ABB RAPID module: Module1

MODULE Module1

    CONST robtarget BackFromStop:=[[674.324181213,-18.678370802,529.462970504],[0.075961249,0.996278649,0.018967815,0.03604114],[-1,-1,-1,1],[9E+09,9E+09,9E+09,9E+09,9E+09,9E+09]];
    CONST robtarget BaseWashers:=[[546.90839525,184.746822368,365.086389723],[0.974259865,-0.054128661,-0.025279397,0.21736779],[0,-1,-3,1],[9E+09,9E+09,9E+09,9E+09,9E+09,9E+09]];
    CONST robtarget Home:=[[667.846096908,0,609.320508076],[0,0.965925826,0,-0.258819045],[0,0,0,0],[9E+09,9E+09,9E+09,9E+09,9E+09,9E+09]];
    CONST robtarget MeasureStationWasher:=[[889,-50,411],[1,0,0,0],[-1,-1,-2,1],[9E+09,9E+09,9E+09,9E+09,9E+09,9E+09]];
    CONST robtarget New_Bin:=[[62.650092384,-476.795876247,452.830737958],[0.710346717,-0.001344528,0.703822969,-0.006241907],[-1,2,-1,1],[9E+09,9E+09,9E+09,9E+09,9E+09,9E+09]];
    CONST robtarget New_GoodStation:=[[883,-346,485.773],[0,0.976296007,-0.216439614,0],[-1,0,-1,1],[9E+09,9E+09,9E+09,9E+09,9E+09,9E+09]];
    CONST robtarget New_OtwGoodMag:=[[792.667,-145.899,472.041],[0.016418462,-0.993578509,0.068839613,0.088279605],[-1,-1,0,1],[9E+09,9E+09,9E+09,9E+09,9E+09,9E+09]];
    CONST robtarget New_OtwReWorkMag:=[[771.510212058,-141.598119308,565.814664694],[0.007964554,-0.997301283,0.068792719,0.024377836],[-1,-1,0,1],[9E+09,9E+09,9E+09,9E+09,9E+09,9E+09]];
    CONST robtarget New_PressStation:=[[893,151,440],[0,1,0,0],[0,0,-1,1],[9E+09,9E+09,9E+09,9E+09,9E+09,9E+09]];
    CONST robtarget New_ReWStation:=[[883,-444,457],[0,1,0,0],[-1,-1,0,1],[9E+09,9E+09,9E+09,9E+09,9E+09,9E+09]];
    CONST robtarget NewWasher:=[[489.319,324.987,300.501],[0.957563012,-0.001006022,0.003342539,0.288202869],[0,0,-3,1],[9E+09,9E+09,9E+09,9E+09,9E+09,9E+09]];
    CONST robtarget OtwBin:=[[615.266405472,-207.002344402,542.863057021],[0.004868374,-0.989612793,0.143612335,-0.004279772],[-1,-1,0,1],[9E+09,9E+09,9E+09,9E+09,9E+09,9E+09]];
    CONST robtarget OtwPressStation:=[[800.688,92.23,462.041],[0.003189563,-0.992840049,-0.078776785,0.089736733],[0,-1,0,1],[9E+09,9E+09,9E+09,9E+09,9E+09,9E+09]];
    CONST robtarget OtwReWorkMag2:=[[741.844,-372.845,593.815],[0.009762059,-0.989387249,0.143021385,0.023716198],[-1,-1,0,1],[9E+09,9E+09,9E+09,9E+09,9E+09,9E+09]];
    CONST robtarget OtwShaft:=[[613.579053498,238.399576686,563.991251443],[0.054444807,0.938983938,0.17600685,-0.290459145],[0,0,-1,0],[9E+09,9E+09,9E+09,9E+09,9E+09,9E+09]];
    CONST robtarget OtwShaft11:=[[683.060149822,348.839006306,569.458244101],[0.00187228,-0.972041282,-0.231482209,0.039347519],[0,0,0,1],[9E+09,9E+09,9E+09,9E+09,9E+09,9E+09]];
    CONST robtarget RotateBackFromWasher1:=[[806.362971574,-45.950756254,415.645475922],[0.000871517,-0.992210216,0.008711474,0.124266798],[-1,-1,0,1],[9E+09,9E+09,9E+09,9E+09,9E+09,9E+09]];
    CONST robtarget ShaftPick12:=[[490,426.542,379.462],[0,0.939692621,0.342020143,0],[0,0,0,1],[9E+09,9E+09,9E+09,9E+09,9E+09,9E+09]];
    CONST robtarget Stop1:=[[891,-49,391],[0,1,0,0],[-1,-1,0,1],[9E+09,9E+09,9E+09,9E+09,9E+09,9E+09]];
    CONST robtarget Stop1GetProduct:=[[891.394778408,-51.173361271,440.2609859],[0.00528652,-0.999941944,0.007674812,-0.005409038],[-1,-1,0,1],[9E+09,9E+09,9E+09,9E+09,9E+09,9E+09]];

VAR num cycleCount := 0;
VAR num cycleCount_Good := 0;
VAR num cycleCount_Shaft := 0;
VAR num cycleCount_Re := 0;
VAR num Goodcol := 0;
VAR num shaftCol := 0;
VAR num ReworkCol := 0;
VAR num washerCol := 0;
VAR num End_of_shaft := 6;
VAR num start :=0;

ENDMODULE
